TYPE AssemblyComSubscribe :
STRUCT
  Request : AssemblyComRequest; // contains booleans that are used to start a specific sequence.
  Equipment : AssemblyComSubscribeEquipment;  // structs for equipment objects which are used by the bridges
END_STRUCT
END_TYPE

(* stored: Version 1.1.0.1
   DUT AssemblyComSubscribe: Id {36c3208d-f7e5-4b69-97c4-df3502351039} *)
